//-----------------------------------------------------------------------------------------
//
//                  			ST_HMI_Screen_Home
//
//							Structure datas page Home HMI 			
//-----------------------------------------------------------------------------------------
//
//Auteur: G.GOETZ
//Création: 21.01.2026
//Dernière modification : 21.01.2026 (G.GOETZ)
//       			
//-----------------------------------------------------------------------------------------
//
//     							Liste des modifications  	
//
// 21.01.2026 (G.GOETZ) -> Création		
//-----------------------------------------------------------------------------------------


TYPE ST_HMI_Screen_Home :
STRUCT

	(** SETUP INT **)
		ix1 : INT ; // ?
	
	(** SETUP FLAG **)
		bx1 : BOOL ; // ?

	(** PROCESS INT **)
		iy1 : INT ; // ?
	
	(** PROCESS FLAG **)
		by1 : BOOL ; // ?
	
END_STRUCT
END_TYPE

(* stored: Version 1.1.0.1, ProductVersion 3.1.4026.17
   DUT ST_HMI_Screen_Home: Id {f0a5e31a-5cbf-4065-881b-bc7201bb1148} *)
